(* PLC project PIDControl.project, Inovance company InoProShop(V1.9.0.1) InoProShop(V1.9.0.1) *)
(* stored: creationDateTime 2025-06-02T20:53:02.3002169, modificationDateTime 2025-06-02T14:54:59.8786 *)

(* AJ Jaworowski 2015-02-22\r\n Following the recipe by Peter Nachtwey\r\n http://www.controlguru.com/wp/p80.html *)
FUNCTION_BLOCK HeatExchanger
  VAR_INPUT
    Kp : REAL;  (* System gain *)
    Pp : REAL;  (* Process time *)
    CO : REAL;  (* Output from controller *)
    Dead_t : REAL;  (* The time before the system responds to the disturbance *)
    C : REAL;  (* Initial steady state value *)
    Sample_time : TIME;
  END_VAR
  VAR_OUTPUT
    PV : REAL;  (* Process value at t1 *)
  END_VAR
  VAR
    now : TIME;
    lastTime : TIME;
    lastPV : REAL := 140.0;
    A : REAL;
    B : REAL;
    delta_t : REAL;
    millis : REAL := 1000.0;
  END_VAR

                  now := GTON.ET;
IF ((now - lastTime) > Sample_time) THEN
	delta_t := TIME_TO_REAL(Sample_time)/millis;
	A := EXP(-delta_t/Pp);
	B := 1.0 - A;
	C := 2.0;
	
	//PV := A * lastPV + B * Kp * CO + C;
	PV := 0.987 * lastPV - 0.00679 * CO + C;
	lastPV := PV;

	lastTime := now;
END_IF;
                
END_FUNCTION_BLOCK

(* AJ Jaworowski 2015-02-23\r\n Following the presentation on\r\n http://openenergymonitor.org/emon/node/2999 *)
FUNCTION_BLOCK HeatExchanger2
  VAR_INPUT
    Heat_In : REAL;  (* In principle a radiator in the room [W] *)
    U : REAL;  (* Thermal conductance [W/K] *)
    TC : REAL;  (* Thermal capacity [J/K], commonly cv, specific heat capacity [J/kgK] *)
    Temp_In : REAL;  (* Start temperature in the room [K] *)
    Temp_Out : REAL;  (* Outside temperature [K] *)
    Sample_time : TIME;
  END_VAR
  VAR_OUTPUT
    Temp : REAL;  (* The resulting room temperature *)
  END_VAR
  VAR
    now : TIME;
    lastTime : TIME := TIME#0ms;
    delta_t : REAL;
    heat_flow : REAL;
    lastTemp : REAL;
    TON_0 : TON;
    TON_1 : TON;
    millis : REAL := 1000.0;
  END_VAR

                  now := GTON.ET;
IF ((now - lastTime) > Sample_time) THEN
	delta_t := TIME_TO_REAL(Sample_time)/millis;
	
	//First calculate net heat
	//Heat_In is our heat source
	//Second term is heat flow depending on temperature difference
	//Obs: At start, set lastTime to start temp Temp_In
	IF lastTime = T#0S THEN
		lastTemp := Temp_In;
	END_IF;
	heat_flow := Heat_In - U * (lastTemp - Temp_Out);
	
	//Second: calculate temperature change due to heat_flow
	Temp := lastTemp + heat_flow * delta_t / TC;
	
	//Update variables for next iteration
	lastTemp := Temp;
	lastTime := now;
END_IF;
                
END_FUNCTION_BLOCK

(* A.J. Jaworowski 2015-02-20\r\nSimulering av en tank med RedBull *)
FUNCTION_BLOCK Tank
  VAR_INPUT
    Process_In : REAL;  (* Flöde in per sekund, testa vad som händer on du matar in 100 *)
    Process_Out : REAL;  (* Flöde ut per sekund, typ 90 *)
    SampleTime : TIME;  (* Uppdateringstid, typ 100ms *)
    Lower_limit : REAL;  (* Tankens lägsta nivå, typ 0 *)
    Upper_limit : REAL;  (* Tankens max nivå, kanske 500 *)
  END_VAR
  VAR_OUTPUT
    Level : REAL;  (* Nivån i tanken *)
  END_VAR
  VAR
    now : TIME;
    lastTime : TIME;
    proc_sum_in : REAL := 0.0;
    proc_sum_out : REAL := 0.0;
    temp : REAL;
    millis : REAL := 1000.0;
    proc_out : REAL;
  END_VAR

                  now := GTON.ET;
IF ((now - lastTime) > SampleTime) THEN
	Level := Level +  TIME_TO_REAL(SampleTime)/millis * (Process_In - Process_Out);
	IF Level < Lower_limit THEN
		Level := Lower_limit;
	ELSIF Level > Upper_limit THEN
		Level := Upper_limit;
	END_IF;
	lastTime := now;
END_IF;
                
END_FUNCTION_BLOCK

(* ***************************************************************\r\n* A simple PID controller for Codesys.\r\n* by Alexander Jaworowski\r\n* Inspiration from https://github.com/br3ttb/Arduino-PID-Library\r\n* https://github.com/alexjaw/PID_controller\r\n* This Library is licensed under a MIT License\r\n\r\n 2015-02-22 Bug fix in the calculation of CO_I.\r\n Added derivative term (d(err)/dt = -d(PV)/dt, i.e.\r\n derivative on measurements\r\n*************************************************************** *)
FUNCTION_BLOCK PID_controller
  VAR_INPUT
    SP : REAL;
    PV : REAL;
    Kc : REAL;
    Ti : REAL;
    Td : REAL;
    SampleTime : TIME;  (* Should be ~0.1 * Tp, Tp : the process time [http://www.controlguru.com/2007/012807.html] *)
    LowerLimit : REAL;
    UpperLimit : REAL;
  END_VAR
  VAR_OUTPUT
    CO : REAL;  (* Controller Output *)
    CO_P : REAL;  (* Prportional term *)
    CO_I : REAL;  (* Integral term *)
    CO_D : REAL;  (* Derivative term *)
  END_VAR
  VAR
    millis : REAL := 1000.0;
    now : TIME := TIME#0ms;
    lastTime : TIME := TIME#0ms;
    err : REAL := 0.0;  (* Process error *)
    lastCO_P : REAL := 0.0;  (* Used for calculation of the derivative term *)
    delta_t : REAL;
    lastPV : REAL := 0.0;
  END_VAR

                  //Check parameters
//Ti division by zero
IF Ti = 0.0 THEN
	Ti := 1.0;
END_IF;

//Update PID parameters every sampleTime
now := GTON.ET;
IF ((now - lastTime) > SampleTime) THEN
	err := SP - PV;
	delta_t := TIME_TO_REAL(SampleTime)/millis;
	CO_P := Kc * err;
	CO_I := CO_I + 1.0/Ti * CO_P * delta_t;
	//Add wind-up for CO_I
	IF CO_I < LowerLimit THEN
		CO_I := LowerLimit;
	ELSIF CO_I > UpperLimit THEN
		CO_I := UpperLimit;
	END_IF;
	
	//Observe that d(err)/dt = d(SP)/dt - d(PV)/dt
	//If SP constant,
	//d(err)/dt = - d(PV)/dt
	//Good: no output spikes
	//Bad: some processes need more aggressive tuning
	IF delta_t <> 0.0 THEN
		CO_D := Td * (PV - lastPV)/delta_t;
	END_IF;
	
	//A different approch would be with a tunable filter
	
	CO := CO_P + CO_I + CO_D;
	//Add wind-up for CO
	IF CO < LowerLimit THEN
		CO := LowerLimit;
	ELSIF CO > UpperLimit THEN
		CO := UpperLimit;
	END_IF;
	
	lastTime := now;
	lastPV := PV;
END_IF;
                
END_FUNCTION_BLOCK

PROGRAM PLC_PRG
  VAR
    PID_control_0 : PID_controller;
    HeatEx2_0 : HeatExchanger2;
    SP : REAL := 300.0;
    Temp_out : REAL := 270.0;
  END_VAR

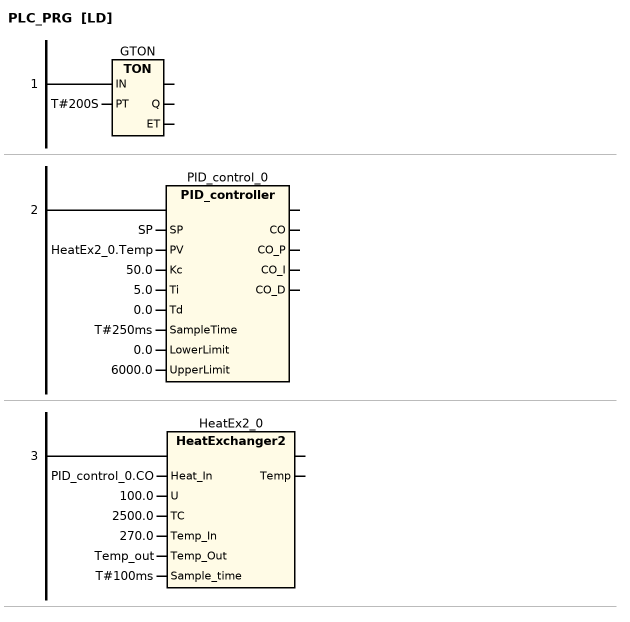
(* LD diagram, written out as Structured Text *)
(* 网络注释 *)

GTON(IN := TRUE, PT := T#200S);
(* 网络注释 *)

PID_control_0(SP := SP, PV := HeatEx2_0.Temp, Kc := 50.0, Ti := 5.0, Td := 0.0, SampleTime := T#250ms, LowerLimit := 0.0, UpperLimit := 6000.0);
(* 网络注释 *)

HeatEx2_0(Heat_In := PID_control_0.CO, U := 100.0, TC := 2500.0, Temp_In := 270.0, Temp_Out := Temp_out, Sample_time := T#100ms);
END_PROGRAM

PROGRAM Test_PID_Heatx
  VAR
    PID_0 : PID_controller;
    Process_out : REAL := 100.0;
    SetPoint : REAL := 20.0;
    A_room_with_a_view : HeatExchanger;
  END_VAR

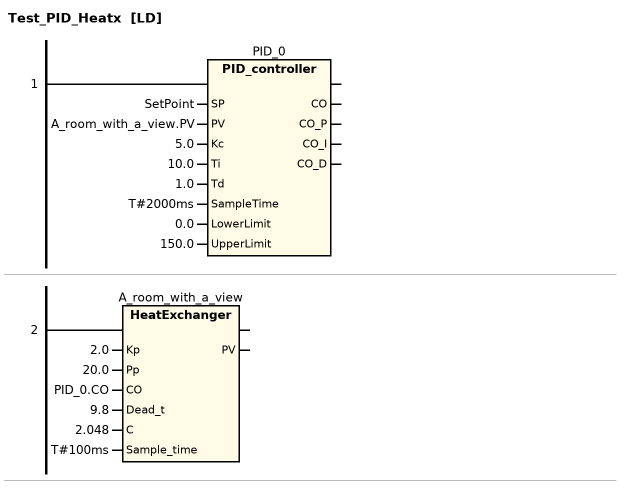
(* LD diagram, written out as Structured Text *)
(* 网络注释 *)

PID_0(SP := SetPoint, PV := A_room_with_a_view.PV, Kc := 5.0, Ti := 10.0, Td := 1.0, SampleTime := T#2000ms, LowerLimit := 0.0, UpperLimit := 150.0);
(* 网络注释 *)

A_room_with_a_view(Kp := 2.0, Pp := 20.0, CO := PID_0.CO, Dead_t := 9.8, C := 2.048, Sample_time := T#100ms);
END_PROGRAM

PROGRAM Test_PID
  VAR
    PID_0 : PID_controller;
    RedBull : Tank;
    Process_out : REAL := 100.0;
    SetPoint : REAL := 250.0;
  END_VAR

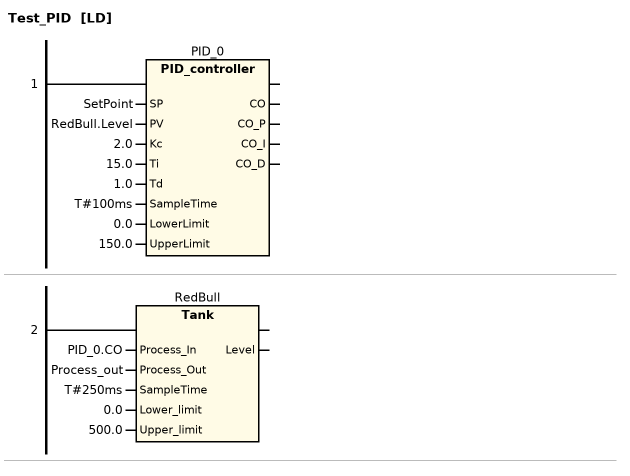
(* LD diagram, written out as Structured Text *)
(* 网络注释 *)

PID_0(SP := SetPoint, PV := RedBull.Level, Kc := 2.0, Ti := 15.0, Td := 1.0, SampleTime := T#100ms, LowerLimit := 0.0, UpperLimit := 150.0);
(* 网络注释 *)

RedBull(Process_In := PID_0.CO, Process_Out := Process_out, SampleTime := T#250ms, Lower_limit := 0.0, Upper_limit := 500.0);
END_PROGRAM

CONFIGURATION Application
  RESOURCE Application ON PLC
    VAR_GLOBAL  (* GVL_Input *)
      Knapp1 : BOOL;  (* Knapp på våning 1 *)
      Knapp2 : BOOL;
      Knapp3 : BOOL;
      Knapp4 : BOOL;
      Vaning1 : BOOL;
      Vaning2 : BOOL;
      Vaning3 : BOOL;
      Vaning4 : BOOL;
      Manuell : BOOL;
      Auto : BOOL;
      Upp : BOOL;
      Ner : BOOL;
      Service_reset : BOOL;
      GTON : TON;
    END_VAR
    VAR_GLOBAL  (* GVL_Output *)
      Lampa1 : BOOL;
      Lampa2 : BOOL;
      Lampa3 : BOOL;
      Lampa4 : BOOL;
      HissUpp : BOOL;
      HissNer : BOOL;
      HissDorr : BOOL;
      LampaAuto : BOOL;
    END_VAR
  END_RESOURCE
END_CONFIGURATION
